// TIA Portal V20 export
TYPE "LER_typePartTrackingCommand"
// stored: Access Published
   STRUCT
      manuLoadDataReq { S7_SetPoint := 'True'} : Bool;
      manuUnloadDataReq : Bool;
      manuDataGenerateReq : Bool;
      manuDataDeleteReq : Bool;
   END_STRUCT;
END_TYPE
